(* CODESYS project waterTankFunctionsAndBlocks_RECOVERED_2026-07-27T13-48-13.project

Project tree, tasks and I/O mapping:
  Device : CODESYS Control Win V3 x64, CODESYS, version 3.5.22.30
    application Application
      libraries: Standard, 3.5.22.0 (System)
      task MainTask (cyclic, interval t#20ms, priority 1) calls PLC_PRG
      function FC_Scaling [LD]
      program PLC_PRG [LD]
*)

// Device/Application/PLC_PRG
PROGRAM PLC_PRG
VAR
	
	Pot1_Fill: REAL;
	Tank1_Fill: REAL;
END_VAR

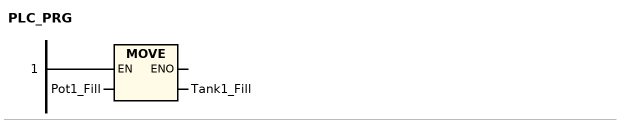
// NETWORK 1
Tank1_Fill := Pot1_Fill;

END_PROGRAM

// Device/Application/FC_Scaling
FUNCTION FC_Scaling : REAL
VAR_INPUT
	Input: REAL;
	Input_Min: REAL;
	Input_Max: REAL;
	Output_Min: REAL;
	Output_Max: REAL;
	
END_VAR
VAR
	Var1: REAL;
	Var2: REAL;
	Var3: REAL;
	Var4: REAL;
	Var5: REAL;
END_VAR

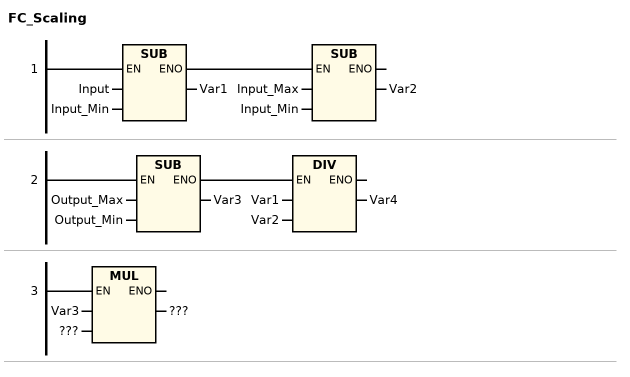
// NETWORK 1
Var1 := Input - Input_Min;
Var2 := Input_Max - Input_Min;

// NETWORK 2
Var3 := Output_Max - Output_Min;
Var4 := Var1 / Var2;

// NETWORK 3
(* Var3 * ???; result not used *)

END_FUNCTION
